PROGRAM MAIN
VAR
END_VAR

END_PROGRAM

(* stored: Version 1.1.0.1
   POU MAIN: Id {3cc89090-40b7-4312-9f84-4c41b4443aa2} *)
